// TIA Portal V19 export
DATA_BLOCK "TOTALIZER DB"   // DB225
{ S7_Optimized_Access := 'TRUE' }
// stored: MemoryReserve 100
   VAR
      BIT : Int;
      "FLOW RATE" : Int;
      "TOTAL FLOW RATE" : Int;
   END_VAR
BEGIN
END_DATA_BLOCK
